(*			
	RafalOS
	Rafał Osajda		29.10.2025		TC 4024.66
	Metody do konfiguracji MAchine control wywoływane z MachineConfigure z pomocą przekazanego ITF
*)
INTERFACE ITF_MCMachineControlConfigure EXTENDS ITF_Base

(*			
	RafalOS
	Rafał Osajda		26.11.2025		TC 4024.66
	Dodawanie szablonu receptury
*)
METHOD PUBLIC AddCreateTemplateFromConfiguration : BOOL
VAR_INPUT
	fbCreateTemplate			: ITF_BaseCreateTemplateOfRecipe;
END_VAR
END_METHOD

(*			
	RafalOS
	Rafał Osajda		13.11.2025		TC 4024.66
	Dodawanie elementów wywoływane z konfiguracji 
*)
METHOD PUBLIC AddElementFromConfiguration : BOOL
VAR_INPUT
	itfElements		: ITF_BaseTopElement;
END_VAR
END_METHOD

(*			
	RafalOS
	Rafał Osajda		13.11.2025		TC 4024.66
	Podpięcie menadżera HMI wywoływane z konfiguracji
*)
METHOD AddHMIManagerFromConfiguration : BOOL
VAR_INPUT
	fbHMIManager			: ITF_BaseGroupElement;
END_VAR
END_METHOD

(*			
	RafalOS
	Rafał Osajda		13.11.2025		TC 4024.66
	Dodanie samego sibie do obsługi w MachineControl
*)
METHOD PUBLIC AddMachineCotrolToYourSelfFromConfiguration : BOOL
VAR_INPUT
END_VAR
END_METHOD

(*			
	RafalOS
	Rafał Osajda		26.11.2025		TC 4024.66
	Dodanie obsługi receptur
*)
METHOD PUBLIC AddModulRecipeFromConfiguration : BOOL
VAR_INPUT
	itfRecipe			: ITF_BaseRecipe;
END_VAR
END_METHOD

(*			
	RafalOS
	Rafał Osajda		13.11.2025		TC 4024.66
	Dodanie modułu sterowania stanami i trybami do machinecontrol z konfiguracji
*)
METHOD PUBLIC AddSaMCotrollerToMachineControlFromConfiguration : BOOL
VAR_INPUT
	itfSaMController			: ITF_SaMController;
END_VAR
END_METHOD

(*			
	RafalOS
	Rafał Osajda		13.11.2025		TC 4024.66
	Wywołanie pierwszego przejścia u wszystkich podzepsołów
*)
METHOD PUBLIC ExecuteFirstCycle : BOOL
VAR_INPUT
END_VAR
END_METHOD

(*			
	RafalOS
	Rafał Osajda		13.11.2025		TC 4024.66
	Zlinkowanie danych wspólnych do dodanych elementów wywoływane z konfiguracji
*)
METHOD PUBLIC LinkCommonDataToAddedElementsFromConfiguration : BOOL
VAR_INPUT
	stCommonData		: REFERENCE TO ST_BaseCommonData;
END_VAR
END_METHOD

(*			
	RafalOS
	Rafał Osajda		13.11.2025		TC 4024.66
	Dodanie głównego komunikatora pomiędzy topelementami do topelementów wywolywane z konfiguracji
*)
METHOD PUBLIC LinkMassangerToaddedTopElementsFromConfiguration : BOOL
VAR_INPUT
	fbCommunicator		: ITF_BaseCommunicator;
END_VAR
END_METHOD

(*			
	RafalOS
	Rafał Osajda		14.11.2025		TC 4024.66
	Podpięcie przyciskow zmiany stanu wywoływane z konfiguracji 
*)
METHOD LinkRequestButtonModeChangeFromConfiguration : BOOL
VAR_INPUT
	iNumberOfRequest			: INT;
	itfRequest					: ITF_MCRequiredChange;
END_VAR
END_METHOD

(*			
	RafalOS
	Rafał Osajda		14.11.2025		TC 4024.66
	Podpięcie przyciskow zmiany trybu i stanu wywoływane z konfiguracji 
*)
METHOD LinkRequestButtonStateChangeFromConfiguration : BOOL
VAR_INPUT
	iNumberOfRequest			: INT;
	itfRequest					: ITF_MCRequiredChange;
END_VAR
END_METHOD

(*			
	RafalOS
	Rafał Osajda		13.11.2025		TC 4024.66
	Podłączenie wsyzstkich zmiennych pochodzących od Programu safety wywoływane w konfiguratorze
*)
METHOD PUBLIC LinkSafetyToaddedElementsFromConfiguration : BOOL
VAR_INPUT
	flSS1				: ITF_BaseFlagGet;
	flSTO				: ITF_BaseFlagGet;
END_VAR
END_METHOD

(*			
	RafalOS
	Rafał Osajda		13.11.2025		TC 4024.66
	Nadanie unikalnych kodów elementom w systemie wywołane z konfiguracji
*)
METHOD PUBLIC SetCodeToAddedElementsFromConfiguration : BOOL
VAR_INPUT
END_VAR
END_METHOD

(*			
	RafalOS
	Rafał Osajda		13.11.2025		TC 4024.66
	Uruchomienie lub wyłączenie obsługi HMI jak jest false fb obsługi nie jest dodawane do MachineControl wywolywane z konfiguracji
*)
METHOD SetEnableHMIServiceFromConfiguration : BOOL
VAR_INPUT
	bValue		: BOOL;
END_VAR
END_METHOD

(*			
	RafalOS
	Rafał Osajda		13.11.2025		TC 4024.66
	Nadaje unikalne ID zgłoszeniom dodanym do elementów w sesyemie wywołane z konfiguracji
*)
METHOD PUBLIC SetIDEventsToAddedElementsFromConfiguration : BOOL
VAR_INPUT
END_VAR
END_METHOD

(*			
	RafalOS
	Rafał Osajda		13.11.2025		TC 4024.66
	Dodanie wszystkim elementom w systemie unikalnego ID
*)
METHOD PUBLIC SetIDToAddedElementsFromConfiguration : BOOL
VAR_INPUT
END_VAR
END_METHOD

(*			
	RafalOS
	Rafał Osajda		14.11.2025		TC 4024.66
	ustawienie trybu poczatkowego wywoływane z konfiguracji
*)
METHOD SetStartModeFromConfiguration : BOOL
VAR_INPUT
	eStartMode				: E_BaseMachineMode;
END_VAR
END_METHOD

END_INTERFACE

(* stored: Version 1.1.0.1
   Itf ITF_MCMachineControlConfigure: Id {407b3a6e-6e4f-4b87-8313-a53f9cca235d}
   Method AddCreateTemplateFromConfiguration: Id {975f47f0-98dd-0dca-2e52-c1e6f55d4f86}
   Method AddElementFromConfiguration: Id {e89dd9da-8dd4-0a9c-2aef-2c77ae2e90a6}
   Method AddHMIManagerFromConfiguration: Id {469471a7-c1b8-090c-0901-f9505ee12d4f}
   Method AddMachineCotrolToYourSelfFromConfiguration: Id {c25f9486-135c-08b4-3ae6-4554d81c2915}
   Method AddModulRecipeFromConfiguration: Id {579798bc-b570-07f3-0ce4-9f9136ef6ddb}
   Method AddSaMCotrollerToMachineControlFromConfiguration: Id {5f46170b-dc51-015c-29c2-1d1aa725f278}
   Method ExecuteFirstCycle: Id {d24ffd5b-ca68-0962-3c0e-990de5787f5e}
   Method LinkCommonDataToAddedElementsFromConfiguration: Id {999c603c-5ddf-0de0-1c6d-967de2690d60}
   Method LinkMassangerToaddedTopElementsFromConfiguration: Id {843efcca-b78f-023a-17c5-679ef58c5dea}
   Method LinkRequestButtonModeChangeFromConfiguration: Id {dcc56f81-e212-0119-324f-69ff5c6b034b}
   Method LinkRequestButtonStateChangeFromConfiguration: Id {63c09a24-b846-0d5b-3dcb-52a59ac8bade}
   Method LinkSafetyToaddedElementsFromConfiguration: Id {c07f7f6a-d91f-08db-2bc2-b870db8dac2e}
   Method SetCodeToAddedElementsFromConfiguration: Id {e29cfd7a-e36e-0ccd-0657-e5130b8e3726}
   Method SetEnableHMIServiceFromConfiguration: Id {040c385a-ca7a-03e1-31b3-f2ce7a8f716f}
   Method SetIDEventsToAddedElementsFromConfiguration: Id {43a66352-c9d0-04a2-24fa-2b0d6136f596}
   Method SetIDToAddedElementsFromConfiguration: Id {243ff86a-db4b-054d-362f-d62d02971187}
   Method SetStartModeFromConfiguration: Id {4c6ccb10-df9b-0976-30d9-7e3c3d75f702} *)
